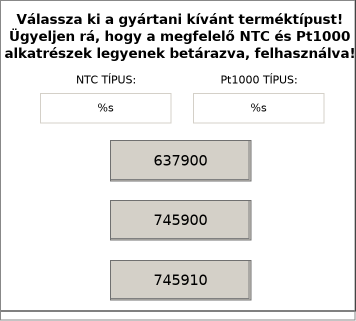
VISUALIZATION Termektipus  // 356x321
    RoundedRectangle (0,0 356x311)
    Label (51,70 110x20), "NTC TÍPUS:"
    Textfield (40,93 131x30), "%s", text variable: GVL.sNTCTypeElozo, colour toggle: GVL.sNTCType='HIBÁS KÓD', input disabled if: true
        OnMouseClick: write GVL.sNTCType via Edit
    Textfield (193,93 131x30), "%s", text variable: GVL.sPtTypeElozo, colour toggle: GVL.sPtType='HIBÁS KÓD', input disabled if: true
        OnMouseClick: write GVL.sPtType via Edit
    Label (204,70 110x20), "Pt1000 TÍPUS:"
    Textfield (120,150 131x30), "%s", text variable: GVL.sProductType, colour toggle: NOT GVL.bProductTypeOK, invisible if: true
        OnMouseClick: write the text variable via Edit
        OnMouseClick: CloseDialog Dialog=Termektipus, Result=OK, NumpadKeypadSet=True
    Button (110,140 141x41), "637900", input disabled if: GVL.UserActual.UserLevel<1
        OnMouseClick: execute { GVL.sProductType:='637900'; }
        OnMouseClick: CloseDialog Dialog=Termektipus, Result=OK, NumpadKeypadSet=True
    Button (110,200 141x40), "745900", input disabled if: GVL.UserActual.UserLevel<1
        OnMouseClick: execute { GVL.sProductType:='745900'; }
        OnMouseClick: CloseDialog Dialog=Termektipus, Result=OK, NumpadKeypadSet=True
    Button (110,260 141x40), "745910", input disabled if: GVL.UserActual.UserLevel<1
        OnMouseClick: execute { GVL.sProductType:='745910'; }
        OnMouseClick: CloseDialog Dialog=Termektipus, Result=OK, NumpadKeypadSet=True
    Label (10,-10 340x93), "Válassza ki a gyártani kívánt terméktípust! Ügyeljen rá, hogy a megfelelő NTC és Pt1000 alkatrészek legyenek betárazva, felhasználva!"
END_VISUALIZATION

(* stored: Version 1.1.0.1, ProductVersion 3.1.4024.11
   Visu Termektipus: Id {e88c6e8f-6913-448a-8d73-890b9800a92a} *)
